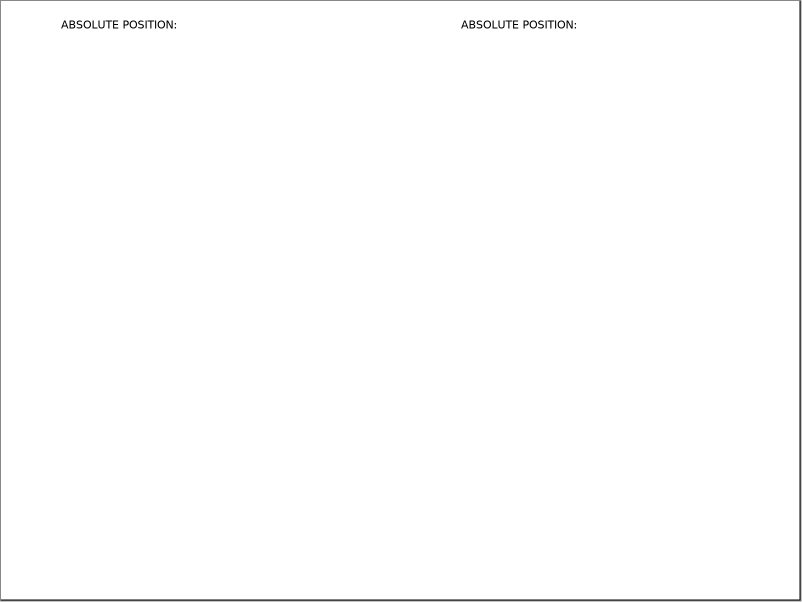
VISUALIZATION F33_Move_Continuous_Absolute  // 802x602
    Rectangle (0,0 800x600)
    Label (10,10 170x30), "ABSOLUTE POSITION:"
    Label (410,10 170x30), "ABSOLUTE POSITION:"
END_VISUALIZATION

(* stored: Version 1.1.0.1, ProductVersion 3.1.4022.7
   Visu F33_Move_Continuous_Absolute: Id {5cc3bfec-b01d-4a42-bb35-aba4c6df19e9} *)
